(* Schneider Machine Expert - Basic project water_pump_from_eight_automation_yt, file version 2.7.0.0 *)
(* ProjectInformations: Name=New project *)

HARDWARE
  Cpu 0: TM221M16R/G
  EthernetConfiguration: NetworkName=M221, IpAllocationMode=FixedAddress, IpAddress=0.0.0.0, SubnetMask=0.0.0.0
  SerialLineConfiguration: Baud=Baud19200, Parity=ParityEven, DataBits=DataBits8, StopBits=StopBits1, PhysicalMedium=PhysicalMediumRs485, TransmissionMode=TransmissionModeModbusRtu, SlaveId=1, Addressing=SlaveAddressing
  MastTask: UsePeriodScanMode=false, PeriodScan=100
  FastTask: Period=255
  CpuBehavior: StartingMode=StartAsPreviousState, AutoSaveRamOnEeprom=true, WatchdogPeriod=250

SYMBOLS  (address, symbol, comment, settings)
  %TM0        [Type=TP, Preset=10, Base=OneSecond]
  %I0.0     STARTING
  %I0.1     LS1
  %I0.2     LS2
  %I0.3     LS3
  %I0.4     TEMP_SWITCH
  %Q0.0     PUMP
  %Q0.1     VALVE1
  %Q0.2     VALVE2
  %Q0.3     MIXER
  %Q0.4     HEATER
  %Q0.5     VALVE3

GRAFCET Grafcet POU
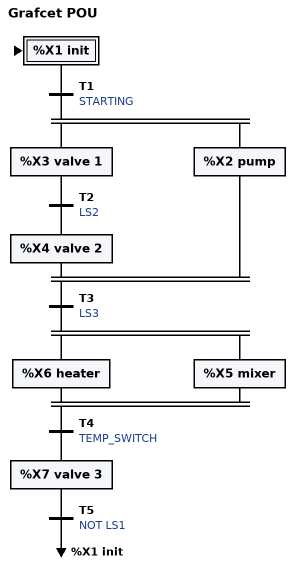
  INITIAL_STEP %X1  (* init *)
  STEP %X2  (* pump *)
  STEP %X3  (* valve 1 *)
  STEP %X4  (* valve 2 *)
  STEP %X5  (* mixer *)
  STEP %X6  (* heater *)
  STEP %X7  (* valve 3 *)
  TRANSITION T1 FROM %X1 TO %X3, %X2 := STARTING;
  TRANSITION T2 FROM %X3 TO %X4 := LS2;
  TRANSITION T3 FROM %X4, %X2 TO %X6, %X5 := LS3;
  TRANSITION T4 FROM %X5, %X6 TO %X7 := TEMP_SWITCH;
  TRANSITION T5 FROM %X7 TO %X1 := NOT LS1;

STEP %X2 pump
  (* SectionNumber=2, StepNumber=2 *)

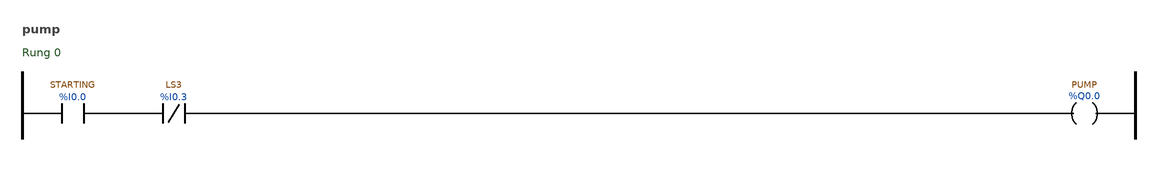

// Rung 0
  LD %I0.0                (* STARTING *)
  ANDN %I0.3              (* LS3 *)
  ST %Q0.0                (* PUMP *)
  // as ST:
  //   PUMP := STARTING AND NOT LS3;

STEP %X3 valve 1
  (* SectionNumber=3, StepNumber=3 *)

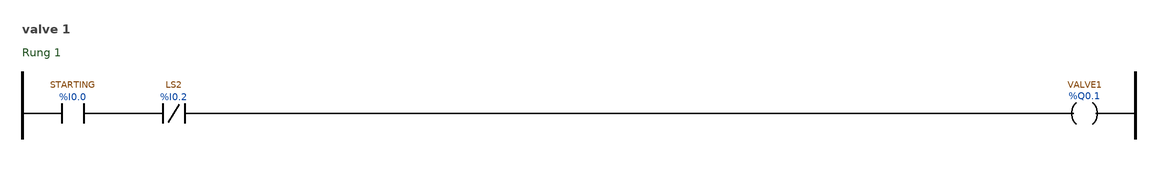

// Rung 1
  LD %I0.0                (* STARTING *)
  ANDN %I0.2              (* LS2 *)
  ST %Q0.1                (* VALVE1 *)
  // as ST:
  //   VALVE1 := STARTING AND NOT LS2;

TRANSITION T1 (%X1 -> %X3, %X2) 
  (* SectionNumber=0 *)

// Rung 2: switch
  LD %I0.0                (* STARTING *)
  ENDT
  // as ST:
  //   TRANSITION := STARTING;

STEP %X4 valve 2
  (* SectionNumber=4, StepNumber=4 *)

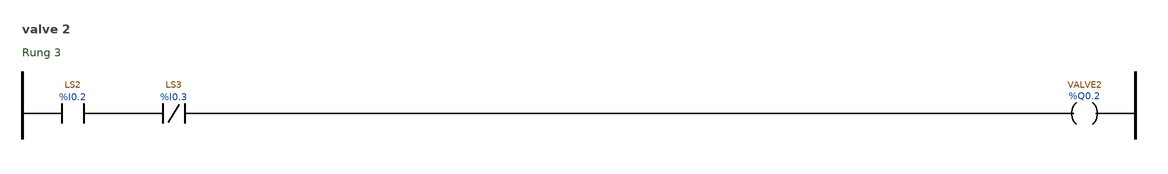

// Rung 3
  LD %I0.2                (* LS2 *)
  ANDN %I0.3              (* LS3 *)
  ST %Q0.2                (* VALVE2 *)
  // as ST:
  //   VALVE2 := LS2 AND NOT LS3;

TRANSITION T2 (%X3 -> %X4) 
  (* SectionNumber=0 *)

// Rung 4: IS-LS2
  LD %I0.2                (* LS2 *)
  ENDT
  // as ST:
  //   TRANSITION := LS2;

STEP %X5 mixer
  (* SectionNumber=5, StepNumber=5 *)

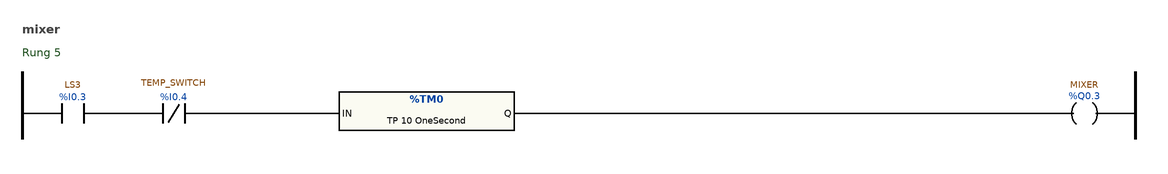

// Rung 5
  BLK %TM0
  LD %I0.3                (* LS3 *)
  ANDN %I0.4              (* TEMP_SWITCH *)
  IN
  OUT_BLK
  LD Q
  ST %Q0.3                (* MIXER *)
  END_BLK
  // as ST:
  //   %TM0(IN := LS3 AND NOT TEMP_SWITCH);
  //   MIXER := %TM0.Q;

STEP %X6 heater
  (* SectionNumber=6, StepNumber=6 *)

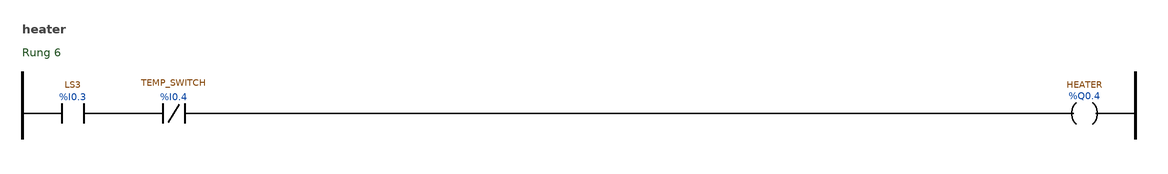

// Rung 6
  LD %I0.3                (* LS3 *)
  ANDN %I0.4              (* TEMP_SWITCH *)
  ST %Q0.4                (* HEATER *)
  // as ST:
  //   HEATER := LS3 AND NOT TEMP_SWITCH;

TRANSITION T3 (%X4, %X2 -> %X6, %X5) 
  (* SectionNumber=0 *)

// Rung 7: is_LS3
  LD %I0.3                (* LS3 *)
  ENDT
  // as ST:
  //   TRANSITION := LS3;

STEP %X7 valve 3
  (* SectionNumber=7, StepNumber=7 *)

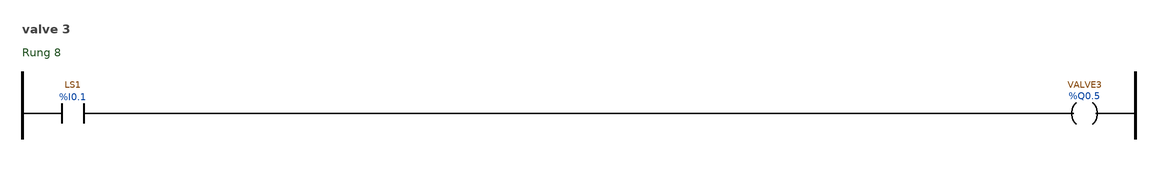

// Rung 8
  LD %I0.1                (* LS1 *)
  ST %Q0.5                (* VALVE3 *)
  // as ST:
  //   VALVE3 := LS1;

TRANSITION T4 (%X5, %X6 -> %X7) 
  (* SectionNumber=0 *)

// Rung 9: temperature switch
  LD %I0.4                (* TEMP_SWITCH *)
  ENDT
  // as ST:
  //   TRANSITION := TEMP_SWITCH;

TRANSITION T5 (%X7 -> %X1) 
  (* SectionNumber=0 *)

// Rung 10: process complete
  LDN %I0.1               (* LS1 *)
  ENDT
  // as ST:
  //   TRANSITION := NOT LS1;
